{attribute 'linkalways'} 
{attribute 'no_explicit_call' := 'This FB is a CLASS and must be accessed using methods or properties'}
{attribute 'enable_dynamic_creation'}
FUNCTION_BLOCK FINAL SUB_BYTE EXTENDS Node
VAR
	in1 : _BYTE(0);
	in2 : _BYTE(0);
	out : _BYTE(0);
END_VAR

METHOD PUBLIC Clone : I_Node
VAR
	pNode : POINTER TO SUB_BYTE;
END_VAR
pNode := __NEW(SUB_BYTE);
Clone := pNode^;
END_METHOD

METHOD FB_init : BOOL
VAR_INPUT
	bInitRetains : BOOL; // if TRUE, the retain variables are initialized (warm start / cold start)
	bInCopyCode : BOOL;  // if TRUE, the instance afterwards gets moved into the copy code (online change)
END_VAR
AddInput('in1',THIS^.in1);
AddInput('in2',THIS^.in2);
AddOutput('out', THIS^.out);
END_METHOD

METHOD PROTECTED OnExecute
VAR
END_VAR
out.Value := in1.Value - in2.Value;
END_METHOD

END_FUNCTION_BLOCK

(* stored: Version 1.1.0.1, ProductVersion 3.1.4024.15
   POU SUB_BYTE: Id {4bee3d61-926c-4695-8040-6333fe521cda}, SpecialFunc None
   Folder Constructor: Id {49e11fb2-e011-4626-ade6-076719936ab9}
   Method Clone: Id {04b1017e-d988-4b27-9b18-d4b1bde63d3d}
   Method FB_init: Id {ab5d38b1-7a46-423b-ae5e-187afa4f29f6}
   Method OnExecute: Id {72c26eb2-9916-4219-b918-1254c420a668} *)
